FUNCTION_BLOCK INTERNAL FINAL FB_WriteRepeatedFieldSInt64Tests EXTENDS FB_TestSuite
VAR_INPUT
END_VAR
VAR_OUTPUT
END_VAR
VAR
    fbFieldCodec : FB_FieldCodecSInt64;
END_VAR

ShouldWriteRepeatedFieldTheory();

METHOD PRIVATE ShouldWriteRepeatedField
VAR_IN_OUT CONSTANT
    aExpected   : ARRAY [*] OF BYTE;
END_VAR
VAR_INPUT
    aValues     : ARRAY [0..7] OF LINT;
    nLength     : UDINT;
    nTag        : UDINT;
    nBufferPosStart     : UDINT;
    nExpectedBufferPos  : UDINT;
    ipFieldCodec        : I_FieldCodec;
END_VAR
VAR_INST
    stState : ST_WriterInternalState;
END_VAR
VAR
    aActualBuffer       : ARRAY [0..63] OF BYTE;
    hr                  : HRESULT;

END_VAR
// Arrange
stState.nBufferPos := nBufferPosStart;
stState.nBufferSize := SIZEOF(aActualBuffer);

// Act
hr := F_WriteRepeatedField(aActualBuffer, stState, anyArray:= F_ToAnyType(aValues), anyFirstElem:= F_ToAnyType(aValues[0]), nLength, F_MakeTag(nTag, E_WireType.LengthDelimited), ipFieldCodec);

// Assert
AssertEquals_DINT(
    Expected:= S_OK,
    Actual:= hr,
    Message:= 'Expected S_OK instead of error');
    
{warning disable C0041}
AssertArrayEquals_BYTE(Expecteds:= aExpected, Actuals:= aActualBuffer, Message:= '');
 
AssertEquals_UDINT(
    Expected:= nExpectedBufferPos,
    Actual:= stState.nBufferPos,
    Message:= CONCAT('Expected stState.nBufferPos to equal ', TO_STRING(nExpectedBufferPos)));
END_METHOD

METHOD PRIVATE ShouldWriteRepeatedFieldTheory : REFERENCE TO FB_Test
VAR CONSTANT
    cRawValueZeroLength     : ARRAY[0..63] OF BYTE := [16#0A, 16#00];
    cRawValue1              : ARRAY[0..63] OF BYTE := [16#00, 16#0A, 16#11, 16#00, 16#A4, 16#13, 16#F2, 16#14, 16#01, 16#F1, 16#14, 16#9C, 16#85, 16#E3, 16#0B, 16#E7, 16#80, 16#80, 16#80, 16#10];  
END_VAR

VAR CONSTANT
    aExpectedZeroLength     : ARRAY [0..7] OF LINT := [0, 0, 0, 0, 0, 0, 0, 0];
    aExpected1              : ARRAY [0..7] OF LINT := [0, 1234, 1337, -1, -1337, 12345678, -2147483700, 0];
END_VAR
TEST(__POUNAME());

ShouldWriteRepeatedField(aExpected:= cRawValueZeroLength, aValues:= aExpectedZeroLength, nLength:= 0, nTag:= 1, nBufferPosStart:= 0, nExpectedBufferPos:= 2, ipFieldCodec:= THIS^.fbFieldCodec);
ShouldWriteRepeatedField(aExpected:= cRawValue1, aValues:= aExpected1, nLength:= 7, nTag:= 1, nBufferPosStart:= 1, nExpectedBufferPos:= 20, ipFieldCodec:= THIS^.fbFieldCodec);

TEST_FINISHED_NAMED(__POUNAME());
END_METHOD

END_FUNCTION_BLOCK

(* stored: Version 1.1.0.1
   POU FB_WriteRepeatedFieldSInt64Tests: Id {649d2692-dd55-40bf-8893-d4981921cebe}, SpecialFunc None
   Method ShouldWriteRepeatedField: Id {3cd3569b-812d-4c6f-b624-0a5ed4988a49}
   Method ShouldWriteRepeatedFieldTheory: Id {18e41782-595a-47ab-abdd-8dc6e67fe676} *)
